FUNCTION_BLOCK differential_protection_4 (* Basic Function Block Type *)
  (* Standard: 61499-2 *)
  (* Version 0.0, 3/23/2016, gulzha, nxtControl GmbH, Template *)
  PACKAGE Main;
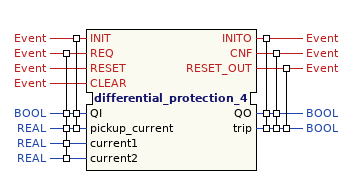
  EVENT_INPUT
    INIT WITH QI, pickup_current; (* Initialization Request *)
    REQ WITH QI, pickup_current, current1, current2; (* Normal Execution Request *)
    RESET;
    CLEAR;
  END_EVENT
  EVENT_OUTPUT
    INITO WITH QO, trip; (* Initialization Confirm *)
    CNF WITH QO, trip; (* Execution Confirmation *)
    RESET_OUT WITH trip;
  END_EVENT
  VAR_INPUT
    QI : BOOL; (* Input event qualifier *)
    pickup_current : REAL;
    current1 : REAL;
    current2 : REAL;
  END_VAR
  VAR_OUTPUT
    QO : BOOL; (* Output event qualifier *)
    trip : BOOL;
  END_VAR
  VAR
    fault : BOOL;
    differential : REAL;
    time2 : BOOL;
  END_VAR
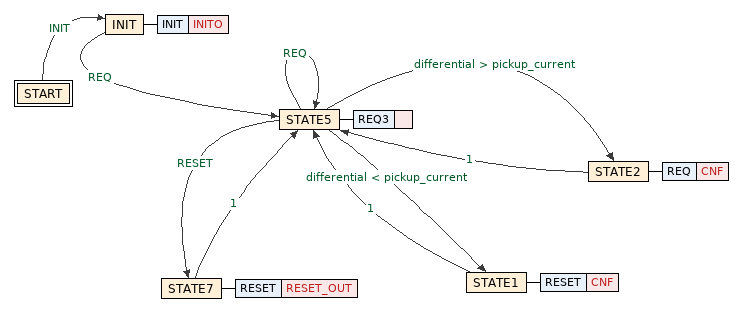
  EC_STATES
    START; (* Initial State *)
    INIT : INIT -> INITO; (* Initialization *)
    STATE2 : REQ -> CNF;
    STATE5 : REQ3;
    STATE7 : RESET -> RESET_OUT;
    STATE1 : RESET -> CNF;
  END_STATES
  EC_TRANSITIONS
    START TO INIT := INIT;
    STATE7 TO STATE5 := 1;
    STATE5 TO STATE7 := RESET;
    STATE5 TO STATE2 := differential > pickup_current;
    STATE5 TO STATE5 := REQ;
    INIT TO STATE5 := REQ;
    STATE2 TO STATE5 := 1;
    STATE5 TO STATE1 := differential < pickup_current;
    STATE1 TO STATE5 := 1;
  END_TRANSITIONS
  ALGORITHM INIT IN ST: (* Initialization algorithm *)
trip := FALSE;
fault := FALSE;
time2 := FALSE;

;
  END_ALGORITHM
  ALGORITHM REQ IN ST: (* Normally executed algorithm *)
trip := TRUE;
;
  END_ALGORITHM
  ALGORITHM RESET IN ST:
trip := FALSE;
fault := FALSE;
time2 := FALSE;

;
  END_ALGORITHM
  ALGORITHM REQ2 IN ST:
fault := TRUE;
;
  END_ALGORITHM
  ALGORITHM REQ3 IN ST:
differential := ABS(current1 - current2);
;
  END_ALGORITHM
  ALGORITHM time2_up IN ST:
time2 := TRUE;
;
  END_ALGORITHM
END_FUNCTION_BLOCK
